{attribute 'linkalways'} 
{attribute 'no_explicit_call' := 'This FB is a CLASS and must be accessed using methods or properties'}
{attribute 'enable_dynamic_creation'}
FUNCTION_BLOCK _TcVnParamsBlobDetection EXTENDS StructuredDatatypeBase
VAR
	localData : TcVnParamsBlobDetection;
	activeData : REFERENCE TO TcVnParamsBlobDetection REF= localData;
    _bFilterByArea         : _BOOL(localdata.bFilterByArea);
    _bFilterByCircularity  : _BOOL(localdata.bFilterByCircularity);
    _bFilterByConvexity    : _BOOL(localdata.bFilterByConvexity);
    _bFilterByEccentricity : _BOOL(localdata.bFilterByEccentricity);
    _bFilterByInertiaRatio : _BOOL(localdata.bFilterByInertiaRatio);
    _fMinArea              : _REAL(localdata.fMinArea);
    _fMaxArea              : _REAL(localdata.fMaxArea);
    _fMinCircularity       : _REAL(localdata.fMinCircularity);
    _fMaxCircularity       : _REAL(localdata.fMaxCircularity);
    _fMinConvexity         : _REAL(localdata.fMinConvexity);
    _fMaxConvexity         : _REAL(localdata.fMaxConvexity);
    _fMinEccentricity      : _REAL(localdata.fMinEccentricity);
    _fMaxEccentricity      : _REAL(localdata.fMaxEccentricity);
    _fMinInertiaRatio      : _REAL(localdata.fMinInertiaRatio);
    _fMaxInertiaRatio      : _REAL(localdata.fMaxInertiaRatio);
    _eThresholdType        : _ETcVnThresholdType(localdata.eThresholdType);
    _fMinThreshold         : _REAL(localdata.fMinThreshold);
    _fMaxThreshold         : _REAL(localdata.fMaxThreshold);
    _fThresholdStep        : _REAL(localdata.fThresholdStep);
    _fMinBlobDistance      : _REAL(localdata.fMinBlobDistance);
    _nMinRepeatability     : _UDINT(localdata.nMinRepeatability);
    _eBlobCombination      : _ETcVnBlobCombination(localdata.eBlobCombination);
END_VAR

PROPERTY PUBLIC Address : PVOID
GET
Address := ADR(activeData);
END_GET
END_PROPERTY

PROPERTY PUBLIC bFilterByArea : REFERENCE TO _BOOL
GET
bFilterByArea REF= _bFilterByArea;
END_GET
END_PROPERTY

PROPERTY PUBLIC bFilterByCircularity : REFERENCE TO _BOOL
GET
bFilterByCircularity REF= _bFilterByCircularity;
END_GET
END_PROPERTY

PROPERTY PUBLIC bFilterByConvexity : REFERENCE TO _BOOL
GET
bFilterByConvexity REF= _bFilterByConvexity;
END_GET
END_PROPERTY

PROPERTY PUBLIC bFilterByEccentricity : REFERENCE TO _BOOL
GET
bFilterByEccentricity REF= _bFilterByEccentricity;
END_GET
END_PROPERTY

PROPERTY PUBLIC bFilterByInertiaRatio : REFERENCE TO _BOOL
GET
bFilterByInertiaRatio REF= _bFilterByInertiaRatio;
END_GET
END_PROPERTY

METHOD PUBLIC ClearReference
VAR_INPUT
END_VAR
activeData REF= localData;
SetMemberReference();
END_METHOD

METHOD PUBLIC Clone : I_Datatype
VAR
    pClone : POINTER TO _TcVnParamsBlobDetection;
END_VAR
pClone := __NEW(_TcVnParamsBlobDetection());
pClone^.Value := Value;
Clone := pClone^;
END_METHOD

PROPERTY PUBLIC eBlobCombination : REFERENCE TO _ETcVnBlobCombination
GET
eBlobCombination REF= _eBlobCombination;
END_GET
END_PROPERTY

PROPERTY PUBLIC eThresholdType : REFERENCE TO _ETcVnThresholdType
GET
eThresholdType REF= _eThresholdType;
END_GET
END_PROPERTY

METHOD FB_init : BOOL
VAR_INPUT
	bInitRetains : BOOL; // if TRUE, the retain variables are initialized (warm start / cold start)
	bInCopyCode : BOOL;  // if TRUE, the instance afterwards gets moved into the copy code (online change)
END_VAR
SetMemberReference();
AddMember('bFilterByArea', _bFilterByArea);
AddMember('bFilterByCircularity', _bFilterByCircularity);
AddMember('bFilterByConvexity', _bFilterByConvexity);
AddMember('bFilterByEccentricity', _bFilterByEccentricity);
AddMember('bFilterByInertiaRatio', _bFilterByInertiaRatio);
AddMember('fMinArea', _fMinArea);
AddMember('fMaxArea', _fMaxArea);
AddMember('fMinCircularity', _fMinCircularity);
AddMember('fMaxCircularity', _fMaxCircularity);
AddMember('fMinConvexity', _fMinConvexity);
AddMember('fMaxConvexity', _fMaxConvexity);
AddMember('fMinEccentricity', _fMinEccentricity);
AddMember('fMaxEccentricity', _fMaxEccentricity);
AddMember('fMinInertiaRatio', _fMinInertiaRatio);
AddMember('fMaxInertiaRatio', _fMaxInertiaRatio);
AddMember('eThresholdType', _eThresholdType);
AddMember('fMinThreshold', _fMinThreshold);
AddMember('fMaxThreshold', _fMaxThreshold);
AddMember('fThresholdStep',  _fThresholdStep);
AddMember('fMinBlobDistance', _fMinBlobDistance);
AddMember('nMinRepeatability', _nMinRepeatability);
AddMember('eBlobCombination', _eBlobCombination);
END_METHOD

PROPERTY PUBLIC fMaxArea : REFERENCE TO _REAL
GET
fMaxArea REF= _fMaxArea;
END_GET
END_PROPERTY

PROPERTY PUBLIC fMaxCircularity : REFERENCE TO _REAL
GET
fMaxCircularity REF= _fMaxCircularity;
END_GET
END_PROPERTY

PROPERTY PUBLIC fMaxConvexity : REFERENCE TO _REAL
GET
fMaxConvexity REF= _fMaxConvexity;
END_GET
END_PROPERTY

PROPERTY PUBLIC fMaxEccentricity : REFERENCE TO _REAL
GET
fMaxEccentricity REF= _fMaxEccentricity;
END_GET
END_PROPERTY

PROPERTY PUBLIC fMaxInertiaRatio : REFERENCE TO _REAL
GET
fMaxInertiaRatio REF= _fMaxInertiaRatio;
END_GET
END_PROPERTY

PROPERTY PUBLIC fMaxThreshold : REFERENCE TO _REAL
GET
fMaxThreshold REF= _fMaxThreshold;
END_GET
END_PROPERTY

PROPERTY PUBLIC fMinArea : REFERENCE TO _REAL
GET
fMinArea REF= _fMinArea;
END_GET
END_PROPERTY

PROPERTY PUBLIC fMinBlobDistance : REFERENCE TO _REAL
GET
fMinBlobDistance REF= _fMinBlobDistance;
END_GET
END_PROPERTY

PROPERTY PUBLIC fMinCircularity : REFERENCE TO _REAL
GET
fMinCircularity REF= _fMinCircularity;
END_GET
END_PROPERTY

PROPERTY PUBLIC fMinConvexity : REFERENCE TO _REAL
GET
fMinConvexity REF= _fMinConvexity;
END_GET
END_PROPERTY

PROPERTY PUBLIC fMinEccentricity : REFERENCE TO _REAL
GET
fMinEccentricity REF= _fMinEccentricity;
END_GET
END_PROPERTY

PROPERTY PUBLIC fMinInertiaRatio : REFERENCE TO _REAL
GET
fMinInertiaRatio REF= _fMinInertiaRatio;
END_GET
END_PROPERTY

PROPERTY PUBLIC fMinThreshold : REFERENCE TO _REAL
GET
fMinThreshold REF= _fMinThreshold;
END_GET
END_PROPERTY

PROPERTY PUBLIC fThresholdStep : REFERENCE TO _REAL
GET
fThresholdStep REF= _fThresholdStep;
END_GET
END_PROPERTY

PROPERTY PUBLIC Identifier : T_MAXSTRING
GET
Identifier := 'TcVnParamsBlobDetection';
END_GET
END_PROPERTY

METHOD PUBLIC MakeReferenceTo
VAR_INPUT
	ReferenceTarget : REFERENCE TO TcVnParamsBlobDetection;
END_VAR
activeData REF= ReferenceTarget;
SetMemberReference();
END_METHOD

PROPERTY PUBLIC nMinRepeatability : REFERENCE TO _UDINT
GET
nMinRepeatability REF= _nMinRepeatability;
END_GET
END_PROPERTY

METHOD PROTECTED SetMemberReference
VAR_INPUT
END_VAR
_bFilterByArea.MakeReferenceTo(activeData.bFilterByArea);
_bFilterByCircularity.MakeReferenceTo(activeData.bFilterByCircularity);
_bFilterByConvexity.MakeReferenceTo(activeData.bFilterByConvexity);
_bFilterByEccentricity.MakeReferenceTo(activeData.bFilterByEccentricity);
_bFilterByInertiaRatio.MakeReferenceTo(activeData.bFilterByInertiaRatio);
_fMinArea.MakeReferenceTo(activeData.fMinArea);
_fMaxArea.MakeReferenceTo(activeData.fMaxArea);
_fMinCircularity.MakeReferenceTo(activeData.fMinCircularity);
_fMaxCircularity.MakeReferenceTo(activeData.fMaxCircularity);
_fMinConvexity.MakeReferenceTo(activeData.fMinConvexity);
_fMaxConvexity.MakeReferenceTo(activeData.fMaxConvexity);
_fMinEccentricity.MakeReferenceTo(activeData.fMinEccentricity);
_fMaxEccentricity.MakeReferenceTo(activeData.fMaxEccentricity);
_fMinInertiaRatio.MakeReferenceTo(activeData.fMinInertiaRatio);
_fMaxInertiaRatio.MakeReferenceTo(activeData.fMaxInertiaRatio);
_eThresholdType.MakeReferenceTo(activeData.eThresholdType);
_fMinThreshold.MakeReferenceTo(activeData.fMinThreshold);
_fMaxThreshold.MakeReferenceTo(activeData.fMaxThreshold);
_fThresholdStep.MakeReferenceTo(activeData.fThresholdStep);
_fMinBlobDistance.MakeReferenceTo(activeData.fMinBlobDistance);
_nMinRepeatability.MakeReferenceTo(activeData.nMinRepeatability);
_eBlobCombination.MakeReferenceTo(activeData.eBlobCombination);
END_METHOD

PROPERTY PUBLIC Size : UDINT
GET
Size := SIZEOF(activeData);
END_GET
END_PROPERTY

METHOD TryMakeReferenceTo : BOOL
VAR_INPUT
	Target : I_Datatype;
END_VAR
VAR
	targetAsStruct : I_StructuredDatatype;
	pTargetData : POINTER TO TcVnParamsBlobDetection;
END_VAR
IF NOT Target.TryResolveAsStructuredDatatype(targetAsStruct) THEN
	RETURN;
END_IF

IF NOT (targetAsStruct.Identifier = Identifier) THEN
	RETURN;
END_IF

pTargetData := Target.Address;
activeData REF= pTargetData^;
SetMemberReference();
TryMakeReferenceTo := TRUE;
END_METHOD

PROPERTY PUBLIC Value : REFERENCE TO TcVnParamsBlobDetection
GET
Value REF= activeData;
END_GET
END_PROPERTY

END_FUNCTION_BLOCK

(* stored: Version 1.1.0.1, ProductVersion 3.1.4024.13
   POU _TcVnParamsBlobDetection: Id {8594d258-0ce0-04df-3c10-f9a88b69e168}, SpecialFunc None
   Folder Core: Id {c1f62570-e884-0ae5-15cd-04be7d72b0ad}
   Folder Customize: Id {6b64b7f4-5191-0965-1b53-ddc9b1f78312}
   Folder Constructor: Id {741d1bfb-87a3-0e0d-2649-9eca8ba7d2d0}
   Folder Protected: Id {ca9f214e-3582-03f5-2d3d-4f2178ae766e}
   Property Address: Id {184a05e8-3b21-0d3a-1df5-4e560ead9efd}
   Get Get: Id {7348c008-8788-08c2-3c69-ac48f5485ed7}
   Property bFilterByArea: Id {14a95bbc-9053-0706-259c-eaa803d69159}
   Get Get: Id {34fe697c-c008-05e9-3f47-b09756577e3a}
   Property bFilterByCircularity: Id {51e00aa2-7825-0eba-352d-46fec66f0dd5}
   Get Get: Id {fd776267-a16a-0354-3b84-8d233e6ae045}
   Property bFilterByConvexity: Id {bd6e709e-0383-0208-1f07-a0dc09a26e6b}
   Get Get: Id {df25fc4b-992a-0bd1-2b2d-5279091600ad}
   Property bFilterByEccentricity: Id {f862b523-24a8-06d2-0548-4bfc2cd8e2e3}
   Get Get: Id {25610988-fe02-0519-227b-2abbab1201e1}
   Property bFilterByInertiaRatio: Id {781e950b-6861-05f8-045e-9f5e7b5a7ac8}
   Get Get: Id {1ad36d93-7469-06ac-2a18-728787c92276}
   Method ClearReference: Id {f8faafdb-cfb6-0fc6-18a4-37f62efdc928}
   Method Clone: Id {a9ebd8fa-efe3-061a-2893-e668fd7e4bc8}
   Property eBlobCombination: Id {d4868f56-73b7-007f-2627-8ca90da59a25}
   Get Get: Id {fb8bb9f1-87d9-059d-3948-c45b72667e33}
   Property eThresholdType: Id {1e22ebb6-f747-0460-33db-722d5573bb41}
   Get Get: Id {1ba210f2-2509-0be3-154c-4faf014b8fd6}
   Method FB_init: Id {5736f6eb-fbfe-0e84-1690-6469c73422fc}
   Property fMaxArea: Id {a5b06ad2-182b-0103-39ab-6bdf6cb5c8fc}
   Get Get: Id {2efc4d76-ca14-01ed-3ee3-70f52cf0a707}
   Property fMaxCircularity: Id {e325fb60-e86d-0013-181a-f3fe67f389fa}
   Get Get: Id {0ee910b5-8cd6-0531-1d82-996659002e11}
   Property fMaxConvexity: Id {12d8def8-0746-0002-1d2d-419d588b00ba}
   Get Get: Id {295da30d-09fc-0c79-3036-5dc99a735ea3}
   Property fMaxEccentricity: Id {13f49679-89ea-04ad-1024-f3b865fbb7b7}
   Get Get: Id {4eb2b678-adf8-0005-0f54-ce5c5fe3bf4c}
   Property fMaxInertiaRatio: Id {c9195a8d-6dcc-0b34-0830-b036fa3bad64}
   Get Get: Id {6ecf644d-c088-0e56-020c-49be970978bd}
   Property fMaxThreshold: Id {a565561b-e72a-062c-2000-7af32b6bb167}
   Get Get: Id {ced25f25-dc44-0385-1975-53cb9755d629}
   Property fMinArea: Id {f1d51fe6-83de-050d-2b5c-a9e2a9c6dda8}
   Get Get: Id {795f1688-f175-0d98-270f-7d781d84359b}
   Property fMinBlobDistance: Id {809e1e7c-2e50-092f-3b81-56c35d3a923e}
   Get Get: Id {e9280434-e6f6-0a3e-21c4-6de15ca7a73c}
   Property fMinCircularity: Id {7ed03f45-c0c6-0645-17ef-60b842f02cbc}
   Get Get: Id {1fc406c6-19e1-02a5-21d3-fa2150481d9d}
   Property fMinConvexity: Id {87a2ee18-17e3-0ba8-13d7-2ef19cfe7372}
   Get Get: Id {71c78752-08b5-015e-27b3-ba79b2c284db}
   Property fMinEccentricity: Id {6ec22a94-b42a-055a-349a-d27295be5d7b}
   Get Get: Id {18c8f106-1e2d-0d03-2478-c4967cf8b69f}
   Property fMinInertiaRatio: Id {e0d2c499-febb-0571-1831-4affee09a9e7}
   Get Get: Id {64373eca-76bc-07b5-2322-27f913d4925a}
   Property fMinThreshold: Id {e3a446fb-869a-0430-00c2-1c954c742888}
   Get Get: Id {dce8c73c-774d-02cd-3940-1714a7919e77}
   Property fThresholdStep: Id {4af8c139-e1fc-08ea-184c-4c27fb29aa14}
   Get Get: Id {ce523aa7-6afd-0527-320d-e0649c609a78}
   Property Identifier: Id {8f6ce571-d797-0403-11f5-7e89f88c7208}
   Get Get: Id {28864b14-4834-0e45-2223-4767383ccf25}
   Method MakeReferenceTo: Id {cd282ba9-a074-0642-0f4f-8eb540da00c8}
   Property nMinRepeatability: Id {7ffb30e0-0b12-07ec-1814-0c97baa4b0ef}
   Get Get: Id {7267a750-1457-0ed9-2b5b-2e8674fd8ff2}
   Method SetMemberReference: Id {71352f94-5833-092a-39f3-6c3646c4abe1}
   Property Size: Id {127a3703-30ae-0b8b-3124-bc08cdc2d0ce}
   Get Get: Id {28596c9a-205f-0443-097d-f3dbb53698da}
   Method TryMakeReferenceTo: Id {0549a965-8e82-01e5-3ebb-21fb6988c977}
   Property Value: Id {eed2a5c5-89bd-02f8-2ec2-0dd6b5c38b54}
   Get Get: Id {a101a024-fd33-098a-0448-ad07d108ae10} *)
